{attribute 'qualified_only'}
{attribute 'strict'}
TYPE enum_switch :
(
	off := 0,
	manual := 1,
	auto := 2
);
END_TYPE

(* stored: Version 1.1.0.1, ProductVersion 3.1.4024.12
   DUT enum_switch: Id {56567bb0-4660-4ea9-b86b-f3afb94e9aa9} *)
